(* CODESYS project RCTU.xml

Project tree, tasks and I/O mapping:
  function block RCTU [LD]
*)

// RCTU
FUNCTION_BLOCK RCTU // Rententive up counter
VAR_INPUT
	CU: BOOL; // Count Up
	RESET: BOOL; // Reset Counter to 0
	PV: WORD; // Counter Limit
	RV: WORD; // Starting Value
END_VAR
VAR_OUTPUT
	Q: BOOL; // Counter reached the Limit
	CV: WORD; // Current Counter Value
END_VAR
VAR
END_VAR
VAR // added by the converter: edge detectors and wires of the graphical bodies
    _rt1 : R_TRIG;
END_VAR

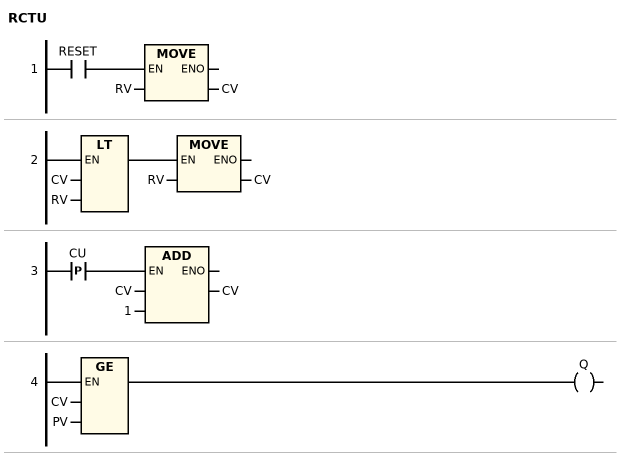
// NETWORK 1
IF RESET THEN CV := RV; END_IF

// NETWORK 2
IF CV < RV THEN CV := RV; END_IF

// NETWORK 3
_rt1(CLK := CU);
IF _rt1.Q THEN CV := CV + 1; END_IF

// NETWORK 4
Q := CV >= PV;

END_FUNCTION_BLOCK
